INTERFACE IXtsTrack

PROPERTY HomePosition : MC_LREAL
GET
END_GET
SET
END_SET
END_PROPERTY

PROPERTY TrackLength : mc_lreal
GET
END_GET
SET
END_SET
END_PROPERTY

END_INTERFACE

(* stored: Version 1.1.0.1, ProductVersion 3.1.4024.12
   Itf IXtsTrack: Id {6f3be1a3-0417-41c4-81da-c6104e06e029}
   Property HomePosition: Id {bc856906-6783-46da-9088-fb5b2100f02f}
   Get Get: Id {68c87207-aac6-470f-970e-e2df3d1317bb}
   Set Set: Id {d1f50dcb-89cb-4cc1-8677-480ae47bbbaf}
   Property TrackLength: Id {c7f52576-ab21-4420-81fd-79b5afa3b103}
   Get Get: Id {fa63afda-8873-4532-879a-f4ddea9e7429}
   Set Set: Id {565c6ca9-71e5-4bda-9e3a-d3e6c8784e36} *)
